TYPE LogEntry :
STRUCT
	Value : STRING;
Datevalue : STRING;
Timevalue : STRING;
	
END_STRUCT
END_TYPE

(* stored: Version 1.1.0.1
   DUT LogEntry: Id {853052ce-d2a1-496f-bef1-a85516dbf24e} *)
